PROGRAM MAIN
VAR
END_VAR

END_PROGRAM

(* stored: Version 1.1.0.1
   POU MAIN: Id {c79c302c-d158-4e42-9b57-27cced6b4588} *)
